RoboDK station: DRILL EXAMPLE.rdk

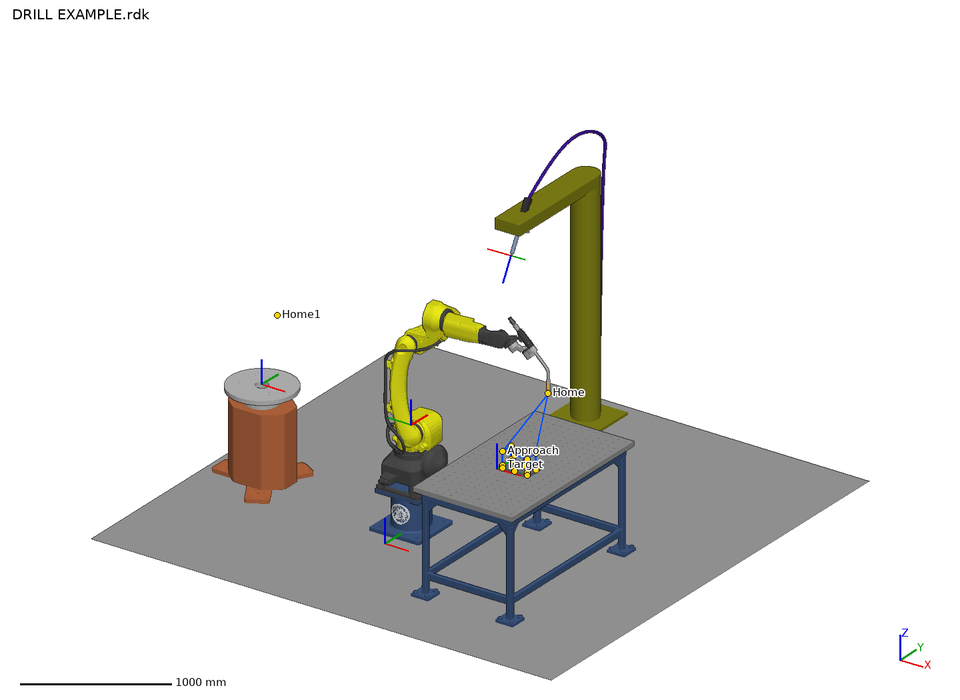
[picture v0: the station drawn from its stored meshes, robots at their saved joint values, targets as dots, program paths as lines]
Station DRILL EXAMPLE (saved by RoboDK 5.9.1). Poses are relative to the parent item; angles as X-Y-Z fixed-axis rotations.
  - frame Fanuc M-10iD/12 Base at (0, 300, 750) mm, rotated rx 0 ry 0 rz 90 deg
    - robot Fanuc M-10iD/12: 6 axes, payload 12 kg, reach 1441 mm, repeatability 0.02 mm, weight 145 kg
        modified DH rows (alpha deg, a mm, theta deg, d mm): 0, 0, 0, 450; -90, 75, -90, 0; 0, 640, 0, 0; -90, 195, 0, 700; 90, 0, 0, 0; -90, 0, 0, 75
        base shift (0, 0, -450) mm
        joint limits [-170, -90, -95, -190, -190, -450] to [170, 160, 180, 190, 190, 450]; home [-87.12, -3.54, 0.98, 0.85, -45.99, 178.78]; saved at [-87.12, -3.54, 0.98, 0.85, -45.99, 178.78]
      - tool Abicor Binzel 45deg Welding Gun, TCP at (0, 0, 400) mm, rotated rx 0 ry 45 rz 0 deg, size 179.1 x 69.8 x 552.4 mm
    - target Home1 (joint target) at (-11.12, 1067.72, 509.95) mm, rotated rx 180 ry 0 rz -90 deg; joints [90.871, -3.548, 0.989, 0.856, -45.995, 178.79] of Fanuc M-10iD/12
    - target Home (joint target) at (48.59, -1066.77, 509.83) mm, rotated rx 179.99 ry 0 rz 92 deg; joints [-87.12, -3.54, 0.98, 0.85, -45.99, 178.78] of Fanuc M-10iD/12
    - target Home (joint target) at (48.59, -1066.77, 509.83) mm, rotated rx 179.99 ry 0 rz 92 deg; joints [-87.12, -3.54, 0.98, 0.85, -45.99, 178.78] of Fanuc M-10iD/12
    - target Home (joint target) at (48.59, -1066.77, 509.83) mm, rotated rx 179.99 ry 0 rz 92 deg; joints [-87.12, -3.54, 0.98, 0.85, -45.99, 178.78] of Fanuc M-10iD/12
  - frame Glue TCP at (0, 1445, 1531) mm, rotated rx -150 ry 0 rz -180 deg
  - frame KUKA KP1-V 500 Base at (-1200, 300, 710) mm
    - robot KUKA KP1-V 500: 1 axes, payload 500 kg
        modified DH rows (alpha deg, a mm, theta deg, d mm): 0, 0, 0, 0
        joint limits [-720] to [720]; home [0]; saved at [0]
    - target P1 (Cartesian target) at (172.52, 117.59, -66.56) mm; joints [0] of KUKA KP1-V 500
  - frame World at (0, 0, 0) mm
    - object Pedestal H12in (Type 1) at (0, 300, 0) mm, size 400 x 400 x 304.8 mm, geometry from Pedestal-H12in-Type-1.sld
    - object Table 1400x800x800mm at (1000, -200, 800) mm, rotated rx 0 ry 0 rz 90 deg, size 1420 x 820 x 800 mm, geometry from Table-1400x800x800mm.sld
    - object Floor at (570, 450, 0) mm, size 3000 x 3000 x 0 mm, geometry from Floor.sld
      - object Floor at (-700, 0, 0) mm, size 3000 x 3000 x 0 mm, geometry from Floor.sld
      - object Floor at (0, 650, 0) mm, size 3000 x 3000 x 0 mm, geometry from Floor.sld
        - object Floor at (-700, 0, 0) mm, size 3000 x 3000 x 0 mm, geometry from Floor.sld
    - object RoboticCell_v1 at (-390, -940, 0) mm, geometry from RoboticCell_v1.step
      - item type 7 RoboticCell_v1-21
      - item type 7 RoboticCell_v1-22
      - item type 7 RoboticCell_v1-23
      - item type 7 RoboticCell_v1-24
      - item type 7 RoboticCell_v1-28
      - item type 7 RoboticCell_v1-29
      - item type 7 RoboticCell_v1-30
      - item type 7 RoboticCell_v1-31
      - item type 7 RoboticCell_v1-32
      - item type 7 RoboticCell_v1-33
      - item type 7 RoboticCell_v1-34
      - item type 7 RoboticCell_v1-35
      - item type 7 RoboticCell_v1-36
      - item type 7 RoboticCell_v1-38
      - item type 7 RoboticCell_v1-46
      - item type 7 RoboticCell_v1-47
      - item type 7 RoboticCell_v1-48
      - item type 7 RoboticCell_v1-27
      - item type 7 RoboticCell_v1-26
      - item type 7 RoboticCell_v1-25
    - object assembly_export at (0, 2300, 0) mm, rotated rx 0 ry 0 rz -180 deg, size 400 x 1136.1 x 2122 mm, geometry from assembly_export.step
    - object Aim Robotics SD 30/55 Dispenser at (0, 1603, 1655) mm, rotated rx -150 ry 0 rz 180 deg, size 63 x 128.2 x 396.5 mm
  - frame CAD_Frame at (900, 0, 800) mm
    - object assembly_export at (0, 0, 0) mm, size 250 x 150 x 25 mm, geometry from assembly_export.step
    - target Approach (Cartesian target) at (25, 25, 125) mm, rotated rx -180 ry 0 rz 92 deg; joints [-87.12, -3.54, 0.98, 0.85, -45.99, 178.78] of Fanuc M-10iD/12
    - target Target (Cartesian target) at (25, 25, 25) mm, rotated rx -180 ry 0 rz 92 deg; joints [-87.12, -3.54, 0.98, 0.85, -45.99, 178.78] of Fanuc M-10iD/12
    - target Drill (Cartesian target) at (25, 25, 5) mm, rotated rx -180 ry 0 rz 92 deg; joints [-87.12, -3.54, 0.98, 0.85, -45.99, 178.78] of Fanuc M-10iD/12
    - target Approach (Cartesian target) at (25, 125, 125) mm, rotated rx -180 ry 0 rz 92 deg; joints [-87.12, -3.54, 0.98, 0.85, -45.99, 178.78] of Fanuc M-10iD/12
    - target Target (Cartesian target) at (25, 125, 25) mm, rotated rx -180 ry 0 rz 92 deg; joints [-87.12, -3.54, 0.98, 0.85, -45.99, 178.78] of Fanuc M-10iD/12
    - target Drill (Cartesian target) at (25, 125, 10) mm, rotated rx -180 ry 0 rz 92 deg; joints [-87.12, -3.54, 0.98, 0.85, -45.99, 178.78] of Fanuc M-10iD/12
    - target Approach (Cartesian target) at (125, 125, 125) mm, rotated rx -180 ry 0 rz 92 deg; joints [-87.12, -3.54, 0.98, 0.85, -45.99, 178.78] of Fanuc M-10iD/12
    - target Target (Cartesian target) at (125, 125, 25) mm, rotated rx -180 ry 0 rz 92 deg; joints [-87.12, -3.54, 0.98, 0.85, -45.99, 178.78] of Fanuc M-10iD/12
    - target Drill (Cartesian target) at (125, 125, 5) mm, rotated rx -180 ry 0 rz 92 deg; joints [-87.12, -3.54, 0.98, 0.85, -45.99, 178.78] of Fanuc M-10iD/12
    - target Approach (Cartesian target) at (125, 25, 125) mm, rotated rx -180 ry 0 rz 92 deg; joints [-87.12, -3.54, 0.98, 0.85, -45.99, 178.78] of Fanuc M-10iD/12
    - target Target (Cartesian target) at (125, 25, 25) mm, rotated rx -180 ry 0 rz 92 deg; joints [-87.12, -3.54, 0.98, 0.85, -45.99, 178.78] of Fanuc M-10iD/12
    - target Drill (Cartesian target) at (125, 25, 5) mm, rotated rx -180 ry 0 rz 92 deg; joints [-87.12, -3.54, 0.98, 0.85, -45.99, 178.78] of Fanuc M-10iD/12
    - target Approach (Cartesian target) at (225, 25, 125) mm, rotated rx -180 ry 0 rz 92 deg; joints [-87.12, -3.54, 0.98, 0.85, -45.99, 178.78] of Fanuc M-10iD/12
    - target Target (Cartesian target) at (225, 25, 25) mm, rotated rx -180 ry 0 rz 92 deg; joints [-87.12, -3.54, 0.98, 0.85, -45.99, 178.78] of Fanuc M-10iD/12
    - target Drill (Cartesian target) at (225, 25, 5) mm, rotated rx -180 ry 0 rz 92 deg; joints [-87.12, -3.54, 0.98, 0.85, -45.99, 178.78] of Fanuc M-10iD/12
    - target Approach (Cartesian target) at (225, 125, 125) mm, rotated rx -180 ry 0 rz 92 deg; joints [-87.12, -3.54, 0.98, 0.85, -45.99, 178.78] of Fanuc M-10iD/12
    - target Target (Cartesian target) at (225, 125, 25) mm, rotated rx -180 ry 0 rz 92 deg; joints [-87.12, -3.54, 0.98, 0.85, -45.99, 178.78] of Fanuc M-10iD/12
    - target Drill (Cartesian target) at (225, 125, 5) mm, rotated rx -180 ry 0 rz 92 deg; joints [-87.12, -3.54, 0.98, 0.85, -45.99, 178.78] of Fanuc M-10iD/12
  - program Drilling (52 instructions, listed below)
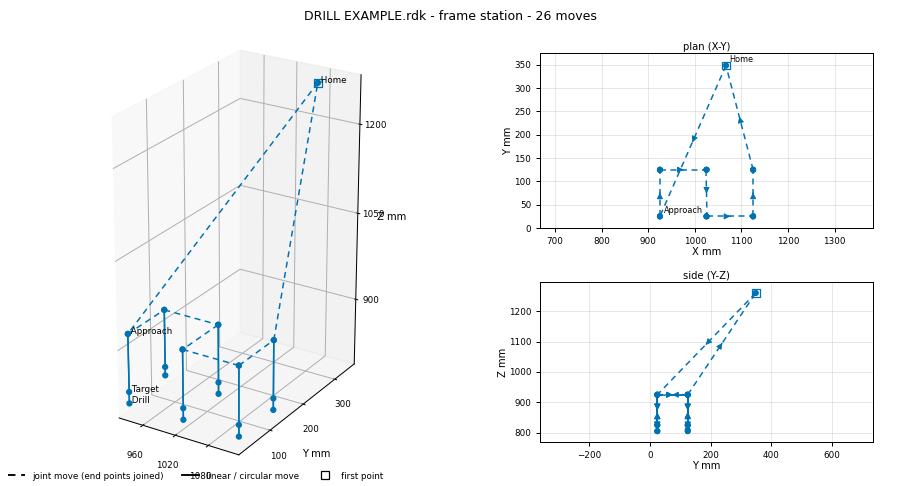
[picture p0: tool path of DRILL EXAMPLE.rdk in frame station, 26 of 26 moves have a stored position in this frame; points joined in program order, loops and branches not executed]

--- program Drilling (robot Fanuc M-10iD/12) ---
  Est. Ref.: CAD_Frame
  Est. herr: Abicor Binzel 45deg Welding Gun
  MoveJ (Home)
  Establecer velocidad (400.0 mm/s)
  MoveJ (Approach)
  Establecer velocidad (80.0 mm/s)
  MoveL (Target)
  Establecer velocidad (20.0 mm/s)
  MoveL (Drill)
  Establecer velocidad (100.0 mm/s)
  MoveL (Approach)
  Establecer velocidad (400.0 mm/s)
  MoveJ (Approach)
  Establecer velocidad (80.0 mm/s)
  MoveL (Target)
  Establecer velocidad (20.0 mm/s)
  MoveL (Drill)
  Establecer velocidad (100.0 mm/s)
  MoveL (Approach)
  Establecer velocidad (400.0 mm/s)
  MoveJ (Approach)
  Establecer velocidad (80.0 mm/s)
  MoveL (Target)
  Establecer velocidad (20.0 mm/s)
  MoveL (Drill)
  Establecer velocidad (100.0 mm/s)
  MoveL (Approach)
  Establecer velocidad (400.0 mm/s)
  MoveJ (Approach)
  Establecer velocidad (80.0 mm/s)
  MoveL (Target)
  Establecer velocidad (20.0 mm/s)
  MoveL (Drill)
  Establecer velocidad (100.0 mm/s)
  MoveL (Approach)
  Establecer velocidad (400.0 mm/s)
  MoveJ (Approach)
  Establecer velocidad (80.0 mm/s)
  MoveL (Target)
  Establecer velocidad (20.0 mm/s)
  MoveL (Drill)
  Establecer velocidad (100.0 mm/s)
  MoveL (Approach)
  Establecer velocidad (400.0 mm/s)
  MoveJ (Approach)
  Establecer velocidad (80.0 mm/s)
  MoveL (Target)
  Establecer velocidad (20.0 mm/s)
  MoveL (Drill)
  Establecer velocidad (100.0 mm/s)
  MoveL (Approach)
  MoveJ (Home)
